{attribute addProperty BoxType "EL3692-0000-0020"}
{attribute addProperty Id "StatusAT %I*Status_5DFF18081621ValueAT %I*DINT32417"}
{attribute addProperty CRC "4256190110"}
{attribute addProperty SizeInBites "48"}
{attribute addProperty SizeInBytes "6"}
TYPE SAI_Inputs_Channel_FDB04E9E :
STRUCT
	{attribute addProperty Name "Status"}
	Status AT %I* : Status_5DFF1808;
	{attribute addProperty Name "Value"}
	Value AT %I* : DINT;
END_STRUCT
END_TYPE

(* stored: Version 1.2.0.0, ProductVersion 3.1.4024.9
   DUT SAI_Inputs_Channel_FDB04E9E: Id {80c5ea47-e01f-4063-8c4b-f54accf95b78} *)
